// TIA Portal V20 export
FUNCTION_BLOCK "FB_FlowMeter_FDH32"   // FB10, LAD
{ S7_Optimized_Access := 'FALSE' }
// Durchfloss-Sensor FD-H Series 
// edited at 17.10.2025
// stored: SetENOAutomatically false
   VAR_INPUT
      iUnscaled_Min : Real;   // 0
      iUnscaled_Max : Real;   // 27648
      iScaled_Flow_Min : Real;
      iFlow_Raw : Int;
      iQuittieren : Bool;   // reset Fehler
      iImpuls : Bool;
      iStoerungUnterdr : Bool;
      iPipe_diameter : Bool;
      iMin_FlowRate : Real;
      iMax_FlowRate : Real;
      iTemp_Raw : Word;
      iScaled_Temp_Min : Real;
      iScaled_Temp_Max : Real;
      iTemp_Above_Limit { ExternalAccessible := 'False'; ExternalVisible := 'False'; ExternalWritable := 'False'} : Real;
      iTemp_Below_limit : Real;
      iErrorFrom_Sensor : Bool;   // Error signal from Sensor
      iAssembly_Place : String;
   END_VAR
   VAR_OUTPUT
      oOutSteo : "UDT_Flowmeter_Stoe";
   END_VAR
   VAR_IN_OUT
      ioVisuSteuern : "UDT_Flowmeter_Steuern";
      ioVisuStatus : "UDT_Flowmeter_Status";
   END_VAR
   VAR
      sFlow_ScaledValue : Real;
      sTemp_ScaledValue : Real;
      Buffer : Array[1..10] of Real;
      Index : DInt;
      Sum : Real;
      sScaled_Max : Real;
      i : Int;
      sAvg : Real;
      sCyclecount : Real;
      sOut_I : Int;
   END_VAR
   VAR_TEMP
      tVKE0 : Bool;
      tVKE1 : Bool;
      tbuffer01 : Int;
      tbuffer02 : Int;
      tbuffer03 : Int;
      tbuffer04 : DInt;
      tbuffer05 : Real;
      tbuffer06 : Word;
      tbuffer07 : Real;
      tNorm_FlowValue : Real;
      tNorm_TempValue : Real;
      tDrahtbruch1 : Bool;
      tDrahtbruch2 : Bool;
      tTempword : Word;
      tFlowword : Word;
      tSecond : Int;
      tMinute : Int;
      tHour : Int;
   END_VAR
   VAR_TEMP   // added for the SCL form of the ladder/FBD networks
      _w1 : Bool;
   END_VAR
BEGIN

REGION Network 1: Create tVKE1 Netzwek
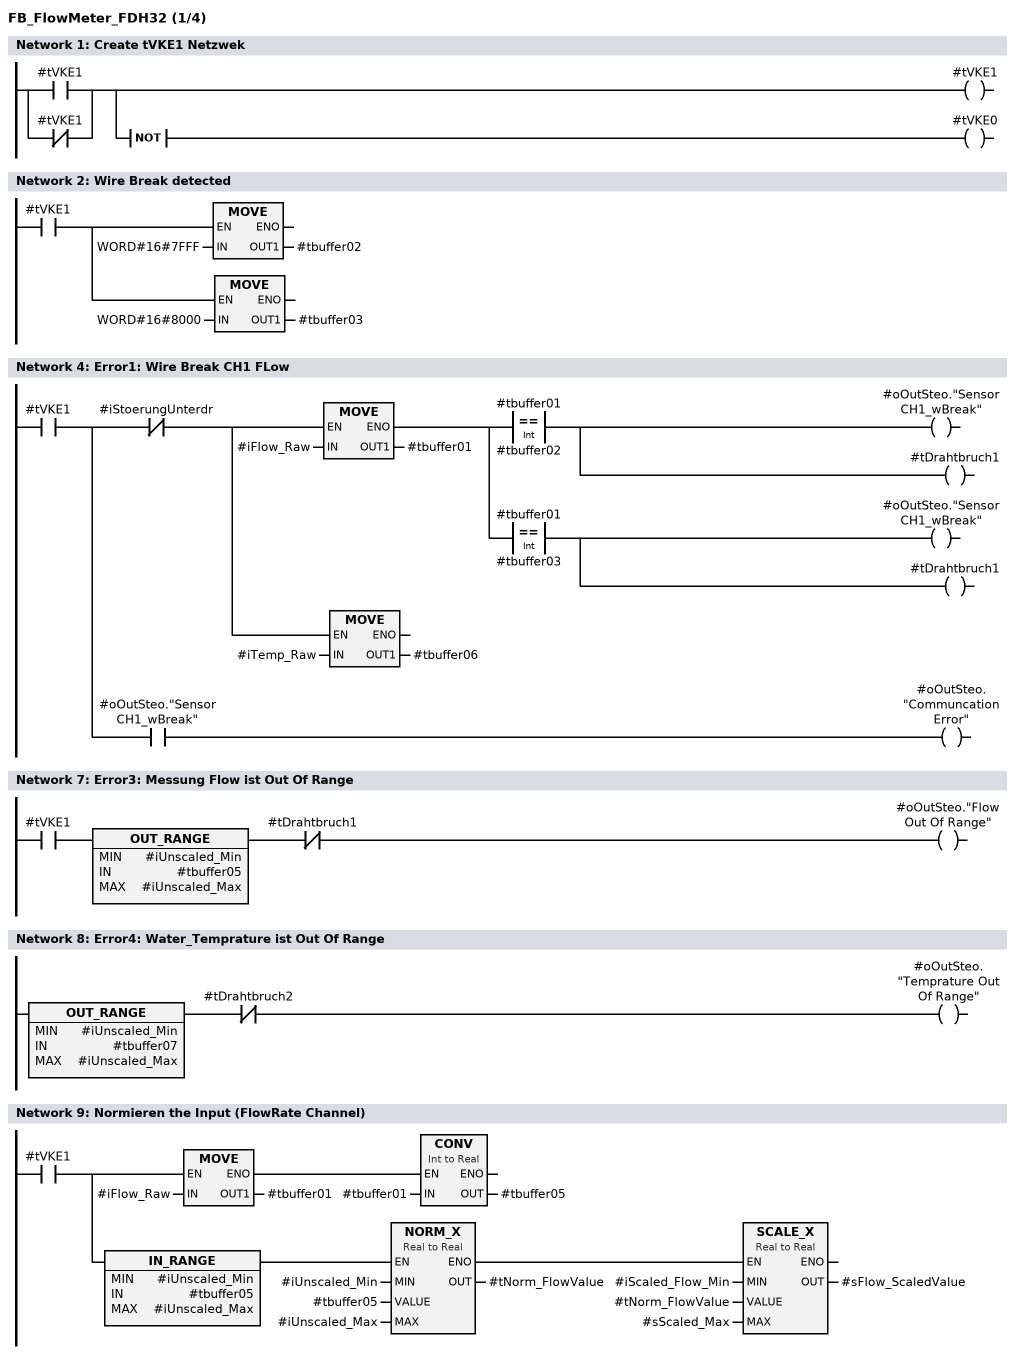
   RUNG wire#powerrail
      Contact( #tVKE1 )
      wire#w1
      Coil( #tVKE1 )
   END_RUNG
   RUNG wire#powerrail
      I_Contact( #tVKE1 )
   END_RUNG wire#w1
   RUNG wire#w1
      Not()
      Coil( #tVKE0 )
   END_RUNG
   // the same network as SCL:
   #tVKE1 := #tVKE1 OR NOT #tVKE1;
   #tVKE0 := NOT #tVKE1;
END_REGION

REGION Network 2: Wire Break detected
   RUNG wire#powerrail
      Contact( #tVKE1 )
      wire#w1
      { S7_GenerateENO := "TRUE" } Move(in := WORD#16#7FFF, out1 => #tbuffer02)
   END_RUNG
   RUNG wire#w1
      { S7_GenerateENO := "TRUE" } Move(in := WORD#16#8000, out1 => #tbuffer03)
   END_RUNG
   // the same network as SCL:
   IF #tVKE1 THEN
       #tbuffer02 := WORD#16#7FFF;
       #tbuffer03 := WORD#16#8000;
   END_IF;
END_REGION

REGION Network 3 (SCL): Reset All Error


   IF #iQuittieren THEN


       #oOutSteo."No Flow Detected"        := 0;
       #oOutSteo."Flow Rate Too Low"       := 0;
       #oOutSteo."Flow Rate Too Hight"     := 0;
       #oOutSteo."Sensor CH1_wBreak"       := 0;
       #oOutSteo."Sensor CH2_wBreak"       := 0;
       #oOutSteo."Temprature Above Limit"  := 0;
       #oOutSteo."Flow Out Of Range"       := 0;
       #oOutSteo."Calibration Error"       := 0;
       #oOutSteo."Air Bubles Detected"     := 0;
       #oOutSteo."Temprature Out Of Range" := 0;
       #oOutSteo."Temprature Below Limit"  := 0;
       #oOutSteo."Reverse Flow Detected"   := 0;
       #oOutSteo."Communcation Error"      := 0;
       #oOutSteo."Clogging or Blockage"    := 0;
       #oOutSteo."Sensor Overheating"      := 0;
       #oOutSteo."Dirty Sensor"            := 0;

   END_IF;
END_REGION

REGION Network 4: Error1: Wire Break CH1 FLow
   RUNG wire#powerrail
      Contact( #tVKE1 )
      wire#w1
      I_Contact( #iStoerungUnterdr )
      wire#w2
      { S7_GenerateENO := "TRUE" } Move(in := #iFlow_Raw, out1 => #tbuffer01)
      wire#w3
      { S7_Templates := "SrcType := Int" } EQ_Contact(in1 := #tbuffer01, in2 := #tbuffer02)
      wire#w4
      Coil( #oOutSteo."Sensor CH1_wBreak" )
   END_RUNG
   RUNG wire#w4
      Coil( #tDrahtbruch1 )
   END_RUNG
   RUNG wire#w3
      { S7_Templates := "SrcType := Int" } EQ_Contact(in1 := #tbuffer01, in2 := #tbuffer03)
      wire#w5
      Coil( #oOutSteo."Sensor CH1_wBreak" )
   END_RUNG
   RUNG wire#w5
      Coil( #tDrahtbruch1 )
   END_RUNG
   RUNG wire#w2
      { S7_GenerateENO := "TRUE" } Move(in := #iTemp_Raw, out1 => #tbuffer06)
   END_RUNG
   RUNG wire#w1
      Contact( #oOutSteo."Sensor CH1_wBreak" )
      Coil( #oOutSteo."Communcation Error" )
   END_RUNG
   // the same network as SCL:
   // ENO of a box is taken as its EN; it also drops when the box reports an error
   #_w1 := #tVKE1 AND NOT #iStoerungUnterdr;
   IF #_w1 THEN #tbuffer01 := #iFlow_Raw; END_IF;
   #oOutSteo."Sensor CH1_wBreak" := #_w1 AND (#tbuffer01 = #tbuffer02);
   #tDrahtbruch1 := #oOutSteo."Sensor CH1_wBreak";
   #oOutSteo."Sensor CH1_wBreak" := #_w1 AND (#tbuffer01 = #tbuffer03);
   #tDrahtbruch1 := #oOutSteo."Sensor CH1_wBreak";
   IF #_w1 THEN #tbuffer06 := #iTemp_Raw; END_IF;
   #oOutSteo."Communcation Error" := #tVKE1 AND #oOutSteo."Sensor CH1_wBreak";
END_REGION

REGION Network 5 (SCL): Evaluate Wire Break CH1 , CH2

   IF #iImpuls AND (#tDrahtbruch1 OR #tDrahtbruch2) THEN
       #tSecond := #tSecond + 1;

       IF #tSecond >= 60 THEN
           #tMinute := #tMinute + 1;
           #tSecond := 0;
       END_IF;

   END_IF;
END_REGION

REGION Network 6 (SCL): Error2: Wire Break CH2 Temprature
   IF #tbuffer06 = #tbuffer02 OR #tbuffer06 = #tbuffer03 THEN
       #tDrahtbruch2 := 1;
       #oOutSteo."Sensor CH2_wBreak" := 1;
   END_IF;
END_REGION

REGION Network 7: Error3: Messung Flow ist Out Of Range
   #oOutSteo."Flow Out Of Range" := #tVKE1 AND ((#tbuffer05 < #iUnscaled_Min) OR (#tbuffer05 > #iUnscaled_Max)) AND NOT #tDrahtbruch1;
END_REGION

REGION Network 8: Error4: Water_Temprature ist Out Of Range
   #oOutSteo."Temprature Out Of Range" := ((#tbuffer07 < #iUnscaled_Min) OR (#tbuffer07 > #iUnscaled_Max)) AND NOT #tDrahtbruch2;
END_REGION

REGION Network 9: Normieren the Input (FlowRate Channel)
   RUNG wire#powerrail
      Contact( #tVKE1 )
      wire#w1
      { S7_GenerateENO := "TRUE" } Move(in := #iFlow_Raw, out1 => #tbuffer01)
      { S7_Templates := "[SrcType := Int, DestType := Real]"; S7_GenerateENO := "TRUE" } Convert(in := #tbuffer01, out => #tbuffer05)
   END_RUNG
   RUNG wire#w1
      { S7_Templates := "SrcType := Real" } InRange(min := #iUnscaled_Min, in := #tbuffer05, max := #iUnscaled_Max)
      { S7_Templates := "[SrcType := Real, DestType := Real]"; S7_GenerateENO := "TRUE" } Normalize(min := #iUnscaled_Min, value := #tbuffer05, max := #iUnscaled_Max, out => #tNorm_FlowValue)
      { S7_Templates := "[SrcType := Real, DestType := Real]"; S7_GenerateENO := "TRUE" } Scale(min := #iScaled_Flow_Min, value := #tNorm_FlowValue, max := #sScaled_Max, out => #sFlow_ScaledValue)
   END_RUNG
   // the same network as SCL:
   // ENO of a box is taken as its EN; it also drops when the box reports an error
   IF #tVKE1 THEN
       #tbuffer01 := #iFlow_Raw;
       #tbuffer05 := INT_TO_REAL(#tbuffer01);
   END_IF;
   IF #tVKE1 AND (#iUnscaled_Min <= #tbuffer05) AND (#tbuffer05 <= #iUnscaled_Max) THEN
       #tNorm_FlowValue := NORM_X(MIN := #iUnscaled_Min, VALUE := #tbuffer05, MAX := #iUnscaled_Max);
       #sFlow_ScaledValue := SCALE_X(MIN := #iScaled_Flow_Min, VALUE := #tNorm_FlowValue, MAX := #sScaled_Max);
   END_IF;
END_REGION

REGION Network 10: Normieren & Scallieren the Water-Temprature
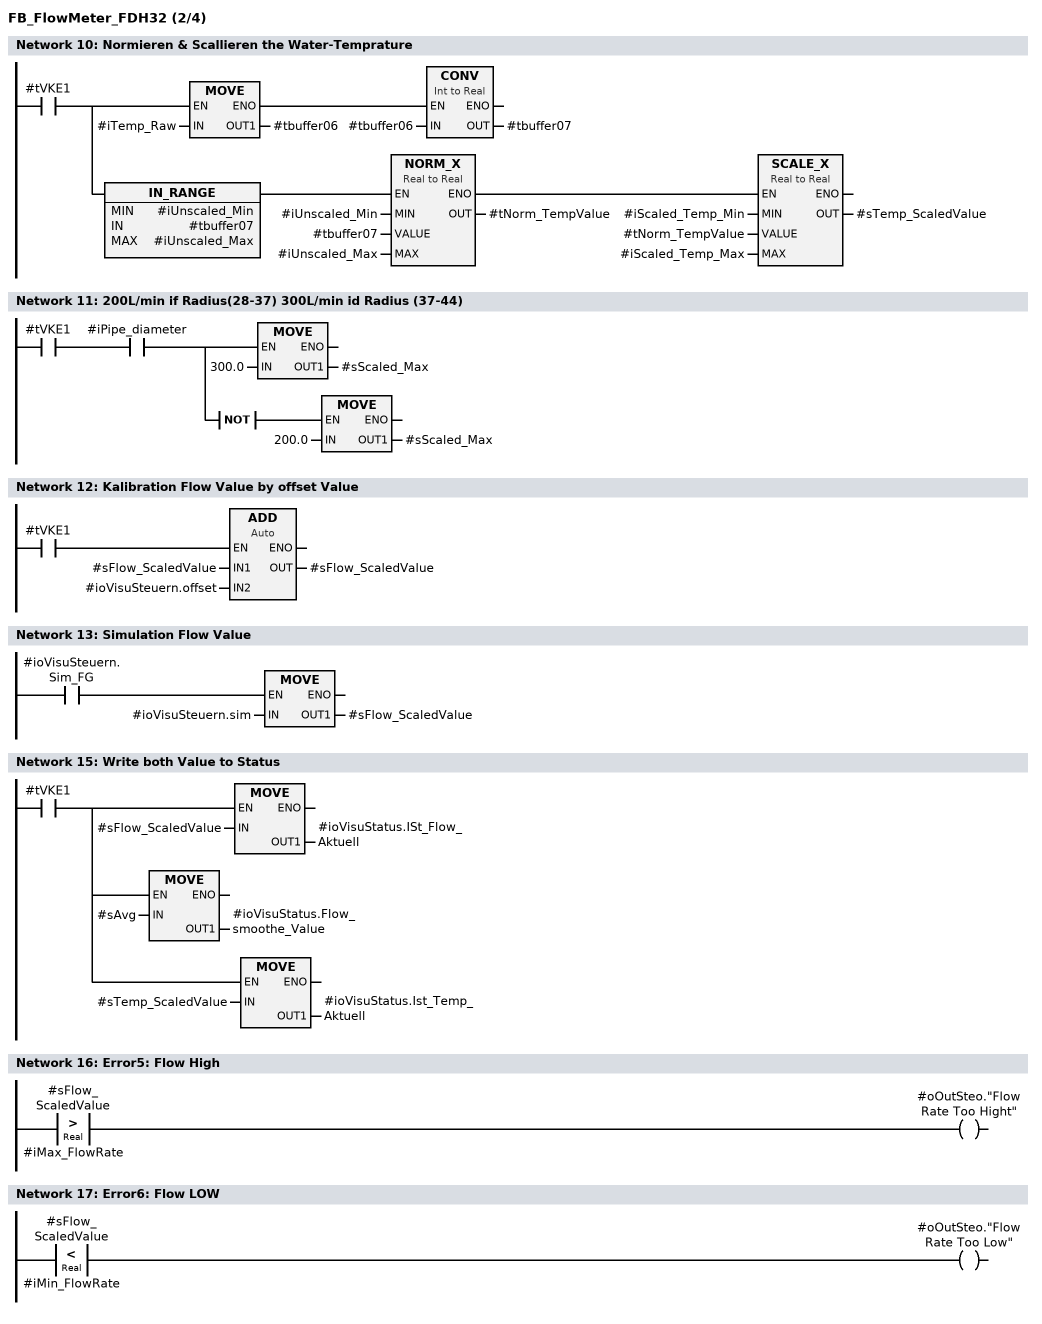
   RUNG wire#powerrail
      Contact( #tVKE1 )
      wire#w1
      { S7_GenerateENO := "TRUE" } Move(in := #iTemp_Raw, out1 => #tbuffer06)
      { S7_Templates := "[SrcType := Int, DestType := Real]"; S7_GenerateENO := "TRUE" } Convert(in := #tbuffer06, out => #tbuffer07)
   END_RUNG
   RUNG wire#w1
      { S7_Templates := "SrcType := Real" } InRange(min := #iUnscaled_Min, in := #tbuffer07, max := #iUnscaled_Max)
      { S7_Templates := "[SrcType := Real, DestType := Real]"; S7_GenerateENO := "TRUE" } Normalize(min := #iUnscaled_Min, value := #tbuffer07, max := #iUnscaled_Max, out => #tNorm_TempValue)
      { S7_Templates := "[SrcType := Real, DestType := Real]"; S7_GenerateENO := "TRUE" } Scale(min := #iScaled_Temp_Min, value := #tNorm_TempValue, max := #iScaled_Temp_Max, out => #sTemp_ScaledValue)
   END_RUNG
   // the same network as SCL:
   // ENO of a box is taken as its EN; it also drops when the box reports an error
   IF #tVKE1 THEN
       #tbuffer06 := #iTemp_Raw;
       #tbuffer07 := INT_TO_REAL(#tbuffer06);
   END_IF;
   IF #tVKE1 AND (#iUnscaled_Min <= #tbuffer07) AND (#tbuffer07 <= #iUnscaled_Max) THEN
       #tNorm_TempValue := NORM_X(MIN := #iUnscaled_Min, VALUE := #tbuffer07, MAX := #iUnscaled_Max);
       #sTemp_ScaledValue := SCALE_X(MIN := #iScaled_Temp_Min, VALUE := #tNorm_TempValue, MAX := #iScaled_Temp_Max);
   END_IF;
END_REGION

REGION Network 11: 200L/min if Radius(28-37) 300L/min id Radius (37-44)
   RUNG wire#powerrail
      Contact( #tVKE1 )
      Contact( #iPipe_diameter )
      wire#w1
      { S7_GenerateENO := "TRUE" } Move(in := 300.0, out1 => #sScaled_Max)
   END_RUNG
   RUNG wire#w1
      Not()
      { S7_GenerateENO := "TRUE" } Move(in := 200.0, out1 => #sScaled_Max)
   END_RUNG
   // the same network as SCL:
   #_w1 := #tVKE1 AND #iPipe_diameter;
   IF #_w1 THEN #sScaled_Max := 300.0; END_IF;
   IF NOT #_w1 THEN #sScaled_Max := 200.0; END_IF;
END_REGION

REGION Network 12: Kalibration Flow Value by offset Value
   RUNG wire#powerrail
      Contact( #tVKE1 )
      { S7_GenerateENO := "TRUE" } Add(in1 := #sFlow_ScaledValue, in2 := #ioVisuSteuern.offset, out => #sFlow_ScaledValue)
   END_RUNG
   // the same network as SCL:
   IF #tVKE1 THEN #sFlow_ScaledValue := #sFlow_ScaledValue + #ioVisuSteuern.offset; END_IF;
END_REGION

REGION Network 13: Simulation Flow Value
   RUNG wire#powerrail
      Contact( #ioVisuSteuern.Sim_FG )
      { S7_GenerateENO := "TRUE" } Move(in := #ioVisuSteuern.sim, out1 => #sFlow_ScaledValue)
   END_RUNG
   // the same network as SCL:
   IF #ioVisuSteuern.Sim_FG THEN #sFlow_ScaledValue := #ioVisuSteuern.sim; END_IF;
END_REGION

REGION Network 14 (SCL): Smoothing the Outsignal
   #sCyclecount := #sCyclecount + 1;

   IF #sCyclecount = 1 THEN
       FOR #i := 1 TO 10 DO
           #Buffer[#i] := #sFlow_ScaledValue;
       END_FOR;

       #Sum := #sFlow_ScaledValue * 10.0;
       #Index := 1;
       #sAvg := #sFlow_ScaledValue;

   ELSE

       #Sum := #Sum - #Buffer[#Index];
       #Buffer[#Index] := #sFlow_ScaledValue;
       #Sum := #Sum + #sFlow_ScaledValue;
       #sAvg := #Sum / 10.0;

       #Index := #Index + 1;
       IF #Index > 10 THEN
           #Index := 1;
       END_IF;
   END_IF;
END_REGION

REGION Network 15: Write both Value to Status
   RUNG wire#powerrail
      Contact( #tVKE1 )
      wire#w1
      { S7_GenerateENO := "TRUE" } Move(in := #sFlow_ScaledValue, out1 => #ioVisuStatus.ISt_Flow_Aktuell)
   END_RUNG
   RUNG wire#w1
      { S7_GenerateENO := "TRUE" } Move(in := #sAvg, out1 => #ioVisuStatus.Flow_smoothe_Value)
   END_RUNG
   RUNG wire#w1
      { S7_GenerateENO := "TRUE" } Move(in := #sTemp_ScaledValue, out1 => #ioVisuStatus.Ist_Temp_Aktuell)
   END_RUNG
   // the same network as SCL:
   IF #tVKE1 THEN
       #ioVisuStatus.ISt_Flow_Aktuell := #sFlow_ScaledValue;
       #ioVisuStatus.Flow_smoothe_Value := #sAvg;
       #ioVisuStatus.Ist_Temp_Aktuell := #sTemp_ScaledValue;
   END_IF;
END_REGION

REGION Network 16: Error5: Flow High
   RUNG wire#powerrail
      { S7_Templates := "SrcType := Real" } GT_Contact(in1 := #sFlow_ScaledValue, in2 := #iMax_FlowRate)
      Coil( #oOutSteo."Flow Rate Too Hight" )
   END_RUNG
   // the same network as SCL:
   #oOutSteo."Flow Rate Too Hight" := #sFlow_ScaledValue > #iMax_FlowRate;
END_REGION

REGION Network 17: Error6: Flow LOW
   RUNG wire#powerrail
      { S7_Templates := "SrcType := Real" } LT_Contact(in1 := #sFlow_ScaledValue, in2 := #iMin_FlowRate)
      Coil( #oOutSteo."Flow Rate Too Low" )
   END_RUNG
   // the same network as SCL:
   #oOutSteo."Flow Rate Too Low" := #sFlow_ScaledValue < #iMin_FlowRate;
END_REGION

REGION Network 18: Error7: Temp High
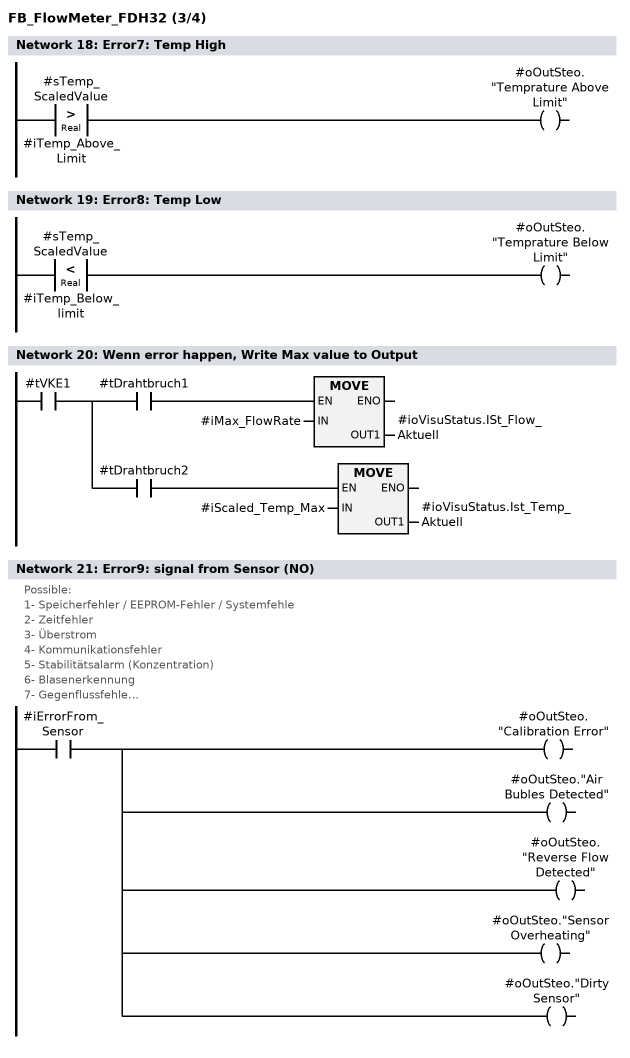
   RUNG wire#powerrail
      { S7_Templates := "SrcType := Real" } GT_Contact(in1 := #sTemp_ScaledValue, in2 := #iTemp_Above_Limit)
      Coil( #oOutSteo."Temprature Above Limit" )
   END_RUNG
   // the same network as SCL:
   #oOutSteo."Temprature Above Limit" := #sTemp_ScaledValue > #iTemp_Above_Limit;
END_REGION

REGION Network 19: Error8: Temp Low
   RUNG wire#powerrail
      { S7_Templates := "SrcType := Real" } LT_Contact(in1 := #sTemp_ScaledValue, in2 := #iTemp_Below_limit)
      Coil( #oOutSteo."Temprature Below Limit" )
   END_RUNG
   // the same network as SCL:
   #oOutSteo."Temprature Below Limit" := #sTemp_ScaledValue < #iTemp_Below_limit;
END_REGION

REGION Network 20: Wenn error happen, Write Max value to Output
   RUNG wire#powerrail
      Contact( #tVKE1 )
      wire#w1
      Contact( #tDrahtbruch1 )
      { S7_GenerateENO := "TRUE" } Move(in := #iMax_FlowRate, out1 => #ioVisuStatus.ISt_Flow_Aktuell)
   END_RUNG
   RUNG wire#w1
      Contact( #tDrahtbruch2 )
      { S7_GenerateENO := "TRUE" } Move(in := #iScaled_Temp_Max, out1 => #ioVisuStatus.Ist_Temp_Aktuell)
   END_RUNG
   // the same network as SCL:
   IF #tVKE1 AND #tDrahtbruch1 THEN #ioVisuStatus.ISt_Flow_Aktuell := #iMax_FlowRate; END_IF;
   IF #tVKE1 AND #tDrahtbruch2 THEN #ioVisuStatus.Ist_Temp_Aktuell := #iScaled_Temp_Max; END_IF;
END_REGION

REGION Network 21: Error9: signal from Sensor (NO)
   // Possible:
   // 1- Speicherfehler / EEPROM-Fehler / Systemfehle
   // 2- Zeitfehler 
   // 3- Überstrom
   // 4- Kommunikationsfehler
   // 5- Stabilitätsalarm (Konzentration)
   // 6- Blasenerkennung
   // 7- Gegenflussfehler
   // 8- Außerhalb des Erkennungsbereichs Temperatur
   RUNG wire#powerrail
      Contact( #iErrorFrom_Sensor )
      wire#w1
      Coil( #oOutSteo."Calibration Error" )
   END_RUNG
   RUNG wire#w1
      Coil( #oOutSteo."Air Bubles Detected" )
   END_RUNG
   RUNG wire#w1
      Coil( #oOutSteo."Reverse Flow Detected" )
   END_RUNG
   RUNG wire#w1
      Coil( #oOutSteo."Sensor Overheating" )
   END_RUNG
   RUNG wire#w1
      Coil( #oOutSteo."Dirty Sensor" )
   END_RUNG
   // the same network as SCL:
   #oOutSteo."Calibration Error" := #iErrorFrom_Sensor;
   #oOutSteo."Air Bubles Detected" := #iErrorFrom_Sensor;
   #oOutSteo."Reverse Flow Detected" := #iErrorFrom_Sensor;
   #oOutSteo."Sensor Overheating" := #iErrorFrom_Sensor;
   #oOutSteo."Dirty Sensor" := #iErrorFrom_Sensor;
END_REGION

REGION Network 22 (SCL): Error_Bit to word
   REGION _BitToWord

       #tFlowword := 0;

       IF #oOutSteo."No Flow Detected" THEN
           #tFlowword := #tFlowword OR W#16#1;
       END_IF;

       IF #oOutSteo."Flow Rate Too Low" THEN
           #tFlowword := #tFlowword OR W#16#2;
       END_IF;

       IF #oOutSteo."Flow Rate Too Hight" THEN
           #tFlowword := #tFlowword OR W#16#4;
       END_IF;

       IF #oOutSteo."Sensor CH1_wBreak" THEN
           #tFlowword := #tFlowword OR W#16#8;
       END_IF;

       IF #oOutSteo."Sensor CH2_wBreak" THEN
           #tFlowword := #tFlowword OR W#16#10;
       END_IF;

       IF #oOutSteo."Temprature Above Limit" THEN
           #tFlowword := #tFlowword OR W#16#20;
       END_IF;

       IF #oOutSteo."Flow Out Of Range" THEN
           #tFlowword := #tFlowword OR W#16#40;
       END_IF;

       IF #oOutSteo."Calibration Error" THEN
           #tFlowword := #tFlowword OR W#16#80;
       END_IF;

       IF #oOutSteo."Air Bubles Detected" THEN
           #tFlowword := #tFlowword OR W#16#100;
       END_IF;

       IF #oOutSteo."Temprature Out Of Range" THEN
           #tFlowword := #tFlowword OR W#16#200;
       END_IF;

       IF #oOutSteo."Temprature Below Limit" THEN
           #tFlowword := #tFlowword OR W#16#400;
       END_IF;

       IF #oOutSteo."Reverse Flow Detected" THEN
           #tFlowword := #tFlowword OR W#16#800;
       END_IF;

       IF #oOutSteo."Communcation Error" THEN
           #tFlowword := #tFlowword OR W#16#1000;
       END_IF;

       IF #oOutSteo."Clogging or Blockage" THEN
           #tFlowword := #tFlowword OR W#16#2000;
       END_IF;

       IF #oOutSteo."Sensor Overheating" THEN
           #tFlowword := #tFlowword OR W#16#4000;
       END_IF;

       IF #oOutSteo."Dirty Sensor" THEN
           #tFlowword := #tFlowword OR W#16#8000;
       END_IF;

       #sOut_I := WORD_TO_INT(#tFlowword);

   END_REGION
END_REGION

REGION Network 23 (SCL): Move Steo to Status

   #ioVisuStatus.MESS_DB_STOE := #tFlowword <> 0;
END_REGION

REGION Network 24 (SCL): Visu Farbe_NO Error

   // No Error  Green
   IF #tFlowword  = 0 THEN
       #ioVisuStatus.VISU_FARBE_Flow := 1;

   END_IF;
END_REGION

REGION Network 25: Visu Farbe_Warning
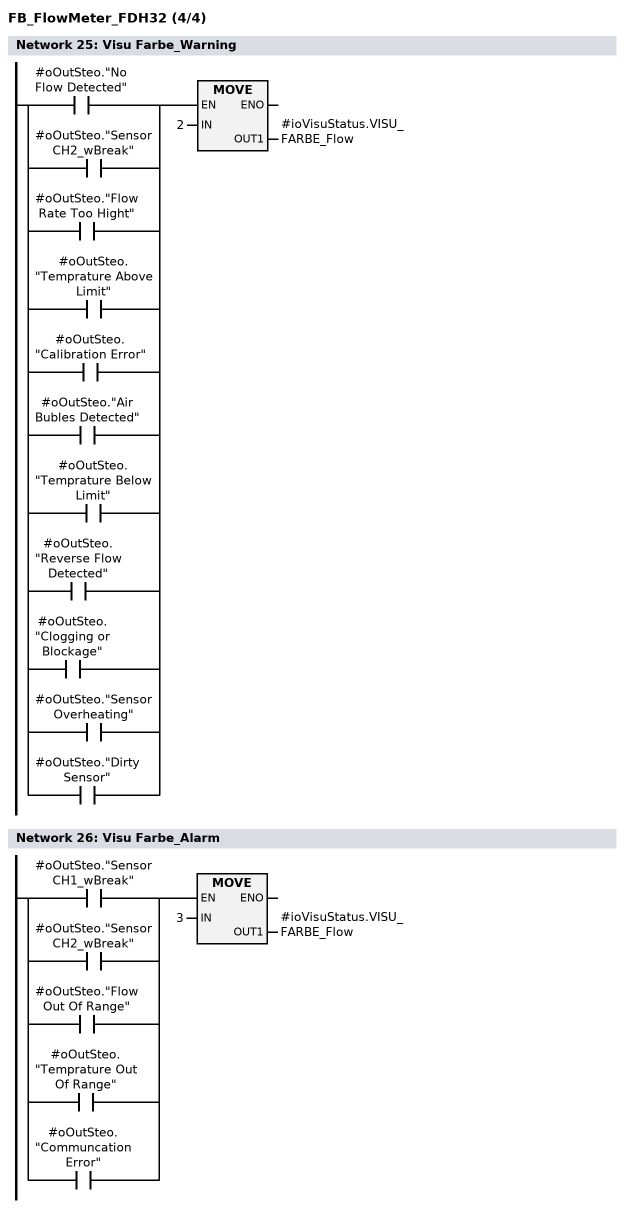
   RUNG wire#powerrail
      Contact( #oOutSteo."No Flow Detected" )
      wire#w1
      { S7_GenerateENO := "TRUE" } Move(in := 2, out1 => #ioVisuStatus.VISU_FARBE_Flow)
   END_RUNG
   RUNG wire#powerrail
      Contact( #oOutSteo."Sensor CH2_wBreak" )
   END_RUNG wire#w1
   RUNG wire#powerrail
      Contact( #oOutSteo."Flow Rate Too Hight" )
   END_RUNG wire#w1
   RUNG wire#powerrail
      Contact( #oOutSteo."Temprature Above Limit" )
   END_RUNG wire#w1
   RUNG wire#powerrail
      Contact( #oOutSteo."Calibration Error" )
   END_RUNG wire#w1
   RUNG wire#powerrail
      Contact( #oOutSteo."Air Bubles Detected" )
   END_RUNG wire#w1
   RUNG wire#powerrail
      Contact( #oOutSteo."Temprature Below Limit" )
   END_RUNG wire#w1
   RUNG wire#powerrail
      Contact( #oOutSteo."Reverse Flow Detected" )
   END_RUNG wire#w1
   RUNG wire#powerrail
      Contact( #oOutSteo."Clogging or Blockage" )
   END_RUNG wire#w1
   RUNG wire#powerrail
      Contact( #oOutSteo."Sensor Overheating" )
   END_RUNG wire#w1
   RUNG wire#powerrail
      Contact( #oOutSteo."Dirty Sensor" )
   END_RUNG wire#w1
   // the same network as SCL:
   IF #oOutSteo."No Flow Detected" OR #oOutSteo."Sensor CH2_wBreak" OR #oOutSteo."Flow Rate Too Hight" OR #oOutSteo."Temprature Above Limit" OR #oOutSteo."Calibration Error" OR #oOutSteo."Air Bubles Detected" OR #oOutSteo."Temprature Below Limit" OR #oOutSteo."Reverse Flow Detected" OR #oOutSteo."Clogging or Blockage" OR #oOutSteo."Sensor Overheating" OR #oOutSteo."Dirty Sensor" THEN
       #ioVisuStatus.VISU_FARBE_Flow := 2;
   END_IF;
END_REGION

REGION Network 26: Visu Farbe_Alarm
   RUNG wire#powerrail
      Contact( #oOutSteo."Sensor CH1_wBreak" )
      wire#w1
      { S7_GenerateENO := "TRUE" } Move(in := 3, out1 => #ioVisuStatus.VISU_FARBE_Flow)
   END_RUNG
   RUNG wire#powerrail
      Contact( #oOutSteo."Sensor CH2_wBreak" )
   END_RUNG wire#w1
   RUNG wire#powerrail
      Contact( #oOutSteo."Flow Out Of Range" )
   END_RUNG wire#w1
   RUNG wire#powerrail
      Contact( #oOutSteo."Temprature Out Of Range" )
   END_RUNG wire#w1
   RUNG wire#powerrail
      Contact( #oOutSteo."Communcation Error" )
   END_RUNG wire#w1
   // the same network as SCL:
   IF #oOutSteo."Sensor CH1_wBreak" OR #oOutSteo."Sensor CH2_wBreak" OR #oOutSteo."Flow Out Of Range" OR #oOutSteo."Temprature Out Of Range" OR #oOutSteo."Communcation Error" THEN
       #ioVisuStatus.VISU_FARBE_Flow := 3;
   END_IF;
END_REGION

REGION Network 27: End Baustein
END_REGION
END_FUNCTION_BLOCK
